// Mitsubishi GX Works2 project: HELLOWORLD270901.gx3   PLC: Q03UDV

PROGRAM MAIN
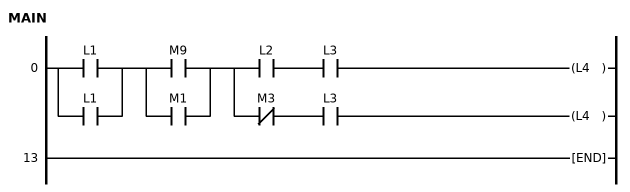
0     LD      L1
      OR      L1
      LD      M9
      OR      M1
      ANB
      MPS
      AND     L2
      AND     L3
      OUT     L4
      MPP
      ANI     M3
      AND     L3
      OUT     L4
13    END
END_PROGRAM
